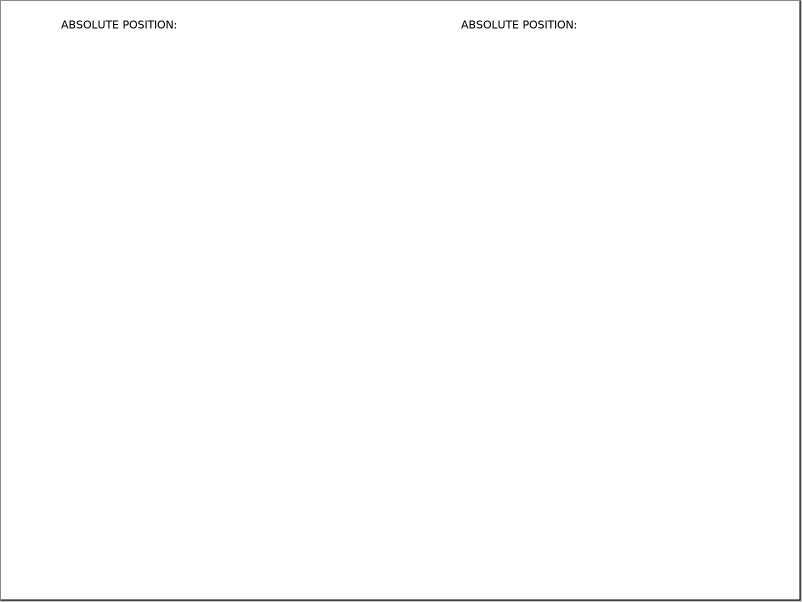
VISUALIZATION F22_Abort_Superposition  // 802x602
    Rectangle (0,0 800x600)
    Label (10,10 170x30), "ABSOLUTE POSITION:"
    Label (410,10 170x30), "ABSOLUTE POSITION:"
END_VISUALIZATION

(* stored: Version 1.1.0.1, ProductVersion 3.1.4022.7
   Visu F22_Abort_Superposition: Id {b752d0a2-1b09-4f5c-904d-230ad86a1a2f} *)
